FUNCTION_BLOCK FB_ToteData
VAR_INPUT
	
END_VAR
VAR_OUTPUT
END_VAR
VAR_IN_OUT
	
END_VAR
VAR
	status	: ToteStatus:= ToteStatus.UNKNOWN;
	barcode	: STRING	:= '';
	barcode_validation	: BarcodeVerificationResult	:= BarcodeVerificationResult.UNVERIFIED;
	
END_VAR

PROPERTY _status : ToteStatus
GET
_status	:= status;
END_GET
SET

status	:= _status;
END_SET
END_PROPERTY

END_FUNCTION_BLOCK

(* stored: Version 1.1.0.1, ProductVersion 3.1.4024.12
   POU FB_ToteData: Id {b550ec73-9a62-494f-ac6c-bd7075901bc6}, SpecialFunc None
   Property _status: Id {a57875de-fbad-45fa-9732-3f1850ab8f1a}
   Get Get: Id {5ed087a4-c79a-4633-8bac-b61050a0ebbb}
   Set Set: Id {dfb0724d-ae07-4d16-9c44-89200ed3f899} *)
